(* PLC project static_torsion.project, CODESYS CODESYS V3.5 SP17 Patch 3 *)
(* stored: creationDateTime 1970-01-01T00:00:00, modificationDateTime 2026-06-22T15:12:39.4699931 *)

CONFIGURATION SoftMotion General Axis Pool
END_CONFIGURATION
